FUNCTION_BLOCK FB_PermIntlk IMPLEMENTS ITF_PermIntlk

VAR
	Name : STRING(Param_PermIntlk.DESCRIPTION_LEN) := 'Permintlk Name';
	Indices : ARRAY[0..(Param_Permintlk.ARRAY_SIZE-1)] OF ST_PermintlkIndex;
	OK : BOOL;
	Message : STRING(Param_PermIntlk.MESSAGE_LEN);
	
	i : USINT;
END_VAR

OK := TRUE;
Message := '';

FOR i :=0 TO (Param_Permintlk.ARRAY_SIZE-1) BY 1 DO 
	IF NOT Indices[i].Condition THEN 
		OK := FALSE;
		IF Message = '' THEN 
			Message := Indices[i].Description;
		ELSE
			Message := CONCAT(CONCAT(Message, ', '),Indices[i].Description);
		END_IF
	END_IF
END_FOR

METHOD M_ClearAll : BOOL
Indices := GVL_PermIntlk.EMPTY_INDICES;
END_METHOD

METHOD M_Set : BOOL
VAR_INPUT
	Index : USINT;
	Description : STRING(Param_PermIntlk.DESCRIPTION_LEN);
	Condition : BOOL;
END_VAR
IF Index < Param_PermIntlk.ARRAY_SIZE THEN 
	Indices[Index].Description := Description;
	Indices[Index].Condition := Condition;
END_IF
END_METHOD

PROPERTY P_Message : STRING(Param_PermIntlk.MESSAGE_LEn)
GET
P_Message := Message;
END_GET
END_PROPERTY

PROPERTY P_Name : STRING(Param_PermIntlk.DESCRIPTION_LEN)
GET
P_Name := Name;
END_GET
SET
Name := P_Name;
END_SET
END_PROPERTY

PROPERTY P_OK : BOOL
GET
P_OK := OK;
END_GET
END_PROPERTY

END_FUNCTION_BLOCK

(* stored: Version 1.1.0.1, ProductVersion 3.1.4024.12
   POU FB_PermIntlk: Id {7fbe70ee-def1-4ef4-a2f4-adfb5314a214}, SpecialFunc None
   Method M_ClearAll: Id {d115b53e-f94d-4dec-8388-59937bb614cc}
   Method M_Set: Id {7d39734a-b77d-4e1a-af5a-41170fe7c770}
   Property P_Message: Id {a87c0be6-f9f8-4fc8-b475-8b8de6405e63}
   Get Get: Id {005e5e77-3125-48b3-a65f-71059b1a0c7d}
   Property P_Name: Id {7743aa23-0f8d-48f4-9584-ccc9f937659b}
   Get Get: Id {cb923d9d-cb30-461f-b781-8320b7a3e8a5}
   Set Set: Id {14c49975-ea7a-4e0f-8ff9-170b1d6371d5}
   Property P_OK: Id {4637f6fe-e1fe-4b37-b0dd-50385ae7316a}
   Get Get: Id {c76fb3a1-23ff-489d-aa12-d938482f1a72} *)
